{attribute 'qualified_only' := ''}
{attribute 'strict' := ''}
TYPE E_SyncConveyorsState :
(
	IDLE := 0,
	RUN := 1,
	FAULT := 10
);
END_TYPE

(* stored: Version 1.1.0.1
   DUT E_SyncConveyorsState: Id {96973905-bd38-49a5-9e33-54f070d5107f} *)
